FUNCTION_BLOCK AXE_plant_FV_Without_NDT (* Basic Function Block Type *)
  (* Standard: 61499-2 *)
  (* Version 0.0, 13/06/2022, Etienne, Schneider Electric, Template *)
  PACKAGE Main;
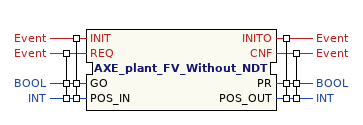
  EVENT_INPUT
    INIT WITH GO, POS_IN; (* Initialization Request *)
    REQ WITH GO, POS_IN; (* Normal Execution Request *)
  END_EVENT
  EVENT_OUTPUT
    INITO WITH PR, POS_OUT; (* Initialization Confirm *)
    CNF WITH PR, POS_OUT; (* Execution Confirmation *)
  END_EVENT
  VAR_INPUT
    GO : BOOL;
    POS_IN : INT;
  END_VAR
  VAR_OUTPUT
    PR : BOOL;
    POS_OUT : INT;
  END_VAR
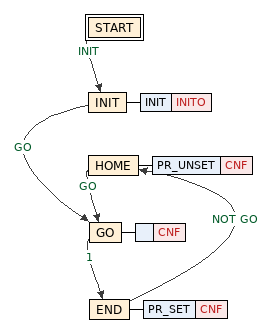
  EC_STATES
    START; (* Initial State *)
    HOME : PR_UNSET -> CNF;
    GO : -> CNF;
    END : PR_SET -> CNF;
    INIT : INIT -> INITO;
  END_STATES
  EC_TRANSITIONS
    HOME TO GO := GO;
    GO TO END := 1;
    END TO HOME := NOT GO;
    START TO INIT := INIT;
    INIT TO GO := GO;
  END_TRANSITIONS
  ALGORITHM INIT IN ST: (* Initialization algorithm *)
;
PR:=FALSE;
  END_ALGORITHM
  ALGORITHM PR_SET IN ST:
;
PR:=TRUE;
POS_OUT:=POS_IN;
  END_ALGORITHM
  ALGORITHM STOP IN ST:
;
PR := FALSE;
POS_OUT:=5;
  END_ALGORITHM
  ALGORITHM PR_UNSET IN ST:
;
PR := FALSE;
  END_ALGORITHM
END_FUNCTION_BLOCK
